FUNCTION_BLOCK FB_SlaveCart
VAR
	
	//Driving force of the car io
	m_driveForce AT %I* :Vec2i;
	
	//stabilizing foot sensor  (normally-closed contact)
	m_stabilizFootSensorLeft AT%I* :BOOL;
	m_stabilizFootSensorRight AT%I* :BOOL;
	m_drivingLeverSensorAuto AT%I* :BOOL;
	m_drivingLeverSensorManual AT%I* :BOOL;
	
	//Trocar IO check
	m_trocarIO AT %I* : ARRAY [1..4] OF UDINT;
	m_trocarCheck : ARRAY [1..4] OF FB_trocarDetect;
	m_trocarFlag : ARRAY [1..4] OF BOOL;
	m_trocarOnFlag : INT:=0;
	
	//output screw break IO 
	m_screwBreak AT %Q* : BOOL;
	m_screwBreakSR : SR;
	
	//car overhang rotation signal is in the arm
	m_carRotaOverhangIO AT%I* : ARRAY [1..4] OF UDINT;
	m_rotaButtonDetect : ARRAY [1..4] OF FB_rotaButtonDetect;
	m_rotaOverhangOnFlag : UDINT :=0;
	
	//cart joint
	m_cartJoints: ARRAY [1..g_cartJntNum] OF FB_CartJoint;
	
	// cart status
	m_cartStatus  : ST_CartStatus;
	
	//cart joint 5 enable detect
	m_standColumnEnableDetect : FB_cartJntEnableDetect;
	m_standColumnDisenableDetect : FB_cartJntDisenableDetect;

	// arm joint data
	m_curMotorPos :Vec8d;
	m_curLinkPos :Vec8d;
	m_curLinkSingle :Vec8d;
	m_curJntPos :Vec8d;
	m_curDHJntPos :Vec6d;
	m_curGripAngle :LREAL;
	m_curJntVel :Vec8d;
	m_curDHJntVel :Vec6d;
	m_curJntTrq :Vec8d;
	m_rawJntCurrent :Vec8d;
	m_filtJntCurrent :Vec8d;
	m_cmdJntTrq :Vec8d;
	m_cmdJntCurrent : Vec8d;
	m_cmdJntPos :Vec8d;
	m_cmdJntVel :Vec8d;

	//SDO Writer
	m_CommunicationCycleInitMZSub1:ARRAY [1..3] OF FB_EcCoESdoWrite;
	m_CommunicationCycleInitMZSub2:ARRAY [1..3] OF FB_EcCoESdoWrite;
	m_CommunicationCycleSub1:INT:=1;
	m_CommunicationCycleSub2:INT:=-3;
	
	//update ui information
	m_joystickSignal:Vec8d;
	m_cartDataFromUI : ST_CartUIData;
	m_ctrlEnable : ST_uiControl;
	m_surgicalStatusF : F_TRIG;
	
	//stand column adjust of setup joint 3
	m_columnJntVel : LREAL;
	m_columnAdjustEnable : BOOL;
	m_limitBufferForCtrl : LREAL := 0.01;
	m_midJntPos : LREAL := 0.1;
	enableTon : ARRAY [1..4] OF FB_TON;
	
	// collision detection
	m_collisionDetection : FB_CartCollisionDetect;
	m_collisionFlag :BOOL:=false;
END_VAR

PROPERTY cartDockingState : UINT
GET
END_GET
SET
m_cartDataFromUI.m_cartDockingState := cartDockingState;
END_SET
END_PROPERTY

PROPERTY cartDrapingState : UINT
GET
END_GET
SET
m_cartDataFromUI.m_cartDrapingState := cartDrapingState;
END_SET
END_PROPERTY

METHOD checkIO : BOOL
VAR_INPUT
END_VAR
VAR
	i:INT;
END_VAR
//check overhang rotation button
m_rotaOverhangOnFlag := MAX( m_rotaButtonDetect[1].run(m_carRotaOverhangIO[1]), m_rotaButtonDetect[2].run(m_carRotaOverhangIO[2]),m_rotaButtonDetect[3].run(m_carRotaOverhangIO[3]),m_rotaButtonDetect[4].run(m_carRotaOverhangIO[4]));

FOR i := 1 TO g_sArmNum BY 1 DO
	//trocar in place monitor
	m_trocarFlag[i] := m_trocarCheck[i].run(m_trocarIO[i] );
END_FOR

m_trocarOnFlag := BOOL_TO_INT(m_trocarFlag[1]) + BOOL_TO_INT(m_trocarFlag[2]) + BOOL_TO_INT(m_trocarFlag[3]) + BOOL_TO_INT(m_trocarFlag[4]);

//setup robot joint 3 adjust and drive column movement
m_columnAdjustEnable :=columnAdjustEnable(o_columnJntVel => m_columnJntVel  );
END_METHOD

PROPERTY cmdJntPos : REFERENCE TO Vec8d
GET
cmdJntPos REF= m_cmdJntPos;
END_GET
END_PROPERTY

PROPERTY cmdJntVel : REFERENCE TO Vec8d
GET
cmdJntVel REF= m_cmdJntVel;
END_GET
END_PROPERTY

METHOD columnAdjustEnable : BOOL
VAR_INPUT
END_VAR

VAR_OUTPUT
	o_columnJntVel : LREAL;
END_VAR

VAR_STAT
	curJntPos : vec4d;
	curJntVel : vec4d;
	columnJntVel : vec4d;
	adjustStartFlag : vec4b;
	m_columnAdjustEnable : vec4b;
END_VAR
VAR
	i : INT;
	armId : INT;
	limitDis : vec4d;
	m_adjustFlag : vec4b;
END_VAR

FOR i := 1 TO g_sArmNum DO
	curJntPos[i] := SetupArmControl.m_setupRobot.m_setupArms[i].m_curJntPos[3];
	curJntVel[i] := SetupArmControl.m_setupRobot.m_setupArms[i].m_curJntVel[3];
	m_adjustFlag[i] := SetupArmControl.m_setupRobot.m_setupArms[i].m_manualAdjustOnFlag AND m_trocarOnFlag=0 AND SetupArmControl.m_setupRobot.m_setupArmState[i] = SetupArmState_ManualAdjust 
									AND NOT SafetyCheck.m_SafetyCheck.m_jntErrFlag[i,0,2] AND NOT SafetyCheck.m_SafetyCheck.m_jntErrFlag[i,0,3] AND NOT SafetyCheck.m_SafetyCheck.m_jntErrFlag[i,3,3] AND NOT SafetyCheck.m_SafetyCheck.m_jntErrFlag[i,2,3] ;
	
	IF m_adjustFlag[i] THEN
		limitDis[i] := MIN(GVL_SetupMotorParameters.g_maxJntPos[i,3] - curJntPos[i], curJntPos[i]-GVL_SetupMotorParameters.g_minJntPos[i,3]);
		IF limitDis[i] < m_limitBufferForCtrl THEN
			adjustStartFlag[i] := TRUE; 
			columnJntVel[i] := sign(m_midJntPos - curJntPos[i]) * GVL_CartControlParameters.g_maxJntVel[5];
		
		ELSIF limitDis[i] >= m_limitBufferForCtrl AND NOT m_columnAdjustEnable[i] THEN
			columnJntVel[i] := 0;
			adjustStartFlag[i] := FALSE;
			
		ELSE
			IF curJntVel[i] <> 0 AND adjustStartFlag[i] THEN
				columnJntVel[i] := -LIMIT(-GVL_CartControlParameters.g_maxJntVel[5], curJntVel[i], GVL_CartControlParameters.g_maxJntVel[5]);
			END_IF
		END_IF
		
		armId := i;
		enableTon[i](IN:= adjustStartFlag[i], PT:= T#3S, Q=> m_columnAdjustEnable[i], ET=> );
		EXIT;
	ELSE
		adjustStartFlag[i] := FALSE;
		columnJntVel[i] := 0;
	END_IF
	enableTon[i](IN:= adjustStartFlag[i], PT:= T#3S, Q=> m_columnAdjustEnable[i], ET=> );
END_FOR

//output stand column joint velocity and start adjust single
IF armId > 0 THEN
	o_columnJntVel := columnJntVel[armId];
END_IF
columnAdjustEnable := m_columnAdjustEnable[1] OR m_columnAdjustEnable[2] OR m_columnAdjustEnable[3] OR m_columnAdjustEnable[4];
END_METHOD

PROPERTY ctrlEnable : REFERENCE TO ST_uiControl
GET
ctrlEnable REF= m_ctrlEnable;
END_GET
SET
END_SET
END_PROPERTY

PROPERTY curDHJntPos :REFERENCE TO Vec6d
GET
curDHJntPos ref= m_curDHJntPos;
END_GET
END_PROPERTY

PROPERTY curDHJntVel :REFERENCE TO Vec6d
GET
curDHJntVel REF= m_curDHJntVel;
END_GET
END_PROPERTY

PROPERTY curJntCurrent :REFERENCE TO Vec8d
GET
curJntCurrent ref=m_filtJntCurrent;
END_GET
END_PROPERTY

PROPERTY curJntPos : REFERENCE TO Vec8d
GET
curJntPos ref=m_curJntPos;
END_GET
END_PROPERTY

PROPERTY curJntVel :REFERENCE TO Vec8d
GET
curJntVel ref=m_curJntVel;
END_GET
END_PROPERTY

PROPERTY curLinkPos :REFERENCE TO Vec8d
GET
curLinkPos ref=m_curLinkPos;
END_GET
END_PROPERTY

PROPERTY curMotorPos : REFERENCE TO  Vec8d
GET
curMotorPos ref=m_curMotorPos;
END_GET
END_PROPERTY

METHOD PUBLIC enable : BOOL
VAR_IN_OUT CONSTANT
	i_jntIdx :Vec8i;
END_VAR
VAR
	i :INT ;
END_VAR
FOR i:=1 TO g_cartJntNum DO
	IF 3<=i AND i<5 THEN
		IF 1= i_jntIdx[i] THEN
			m_cartJoints[i].enableMZ();
		ELSE
			m_cartJoints[i].disable();
		END_IF
	ELSIF i = 5 THEN
		IF 1= i_jntIdx[i] THEN
			m_screwBreak := m_standColumnEnableDetect.run(IOValue:= m_cartJoints[i].enableMZ());
			m_standColumnDisenableDetect.run(IOValue:=FALSE );
		ELSE
			m_standColumnEnableDetect.run(IOValue:= FALSE);
			m_screwBreak :=  NOT m_standColumnDisenableDetect.run(IOValue:=m_cartJoints[i].disable());
		END_IF
	ELSE
		IF 1= i_jntIdx[i] THEN
			m_cartJoints[i].enable();
		ELSE
			m_cartJoints[i].disable();
		END_IF
	END_IF
END_FOR
END_METHOD

METHOD init : BOOL
VAR_INPUT
END_VAR
VAR
	i:INT;
END_VAR


// cart joint init
FOR i:= 1 TO g_cartJntNum BY 1 DO
	m_cartJoints[i].init(i, g_cartCtrlCycleTime);
END_FOR


// joint init
FOR i:=1 TO g_cartJntNum DO
	m_cartJoints[i].initJntPos();
END_FOR


// update cart status if joint position is re-init
updateStatus();



//MingZhi drive example Initialize the communication period
FOR i := 1 TO 3 BY 1 DO
	m_CommunicationCycleInitMZSub1[i](sNetID:= GVL_CartJointEncoderCaliData.g_slaveCartNetID,
				nSlaveAddr := GVL_CartJointEncoderCaliData.g_slaveCartJointNetPort[i+2],
				nSubIndex:=1,nIndex:=16#60C2,pSrcBuf:=ADR(m_CommunicationCycleSub1),cbBufLen:=SIZEOF(m_CommunicationCycleSub1),bExecute:=TRUE);
	
	IF NOT m_CommunicationCycleInitMZSub1[i].bBusy THEN
		m_CommunicationCycleInitMZSub1[i](bExecute:=FALSE);
	END_IF
					
	m_CommunicationCycleInitMZSub2[i](sNetID:= GVL_CartJointEncoderCaliData.g_slaveCartNetID,
					nSlaveAddr := GVL_CartJointEncoderCaliData.g_slaveCartJointNetPort[i+2],
					nSubIndex:=2,nIndex:=16#60C2,pSrcBuf:=ADR(m_CommunicationCycleSub2),cbBufLen:=SIZEOF(m_CommunicationCycleSub2),bExecute:=TRUE);
	
	IF NOT m_CommunicationCycleInitMZSub2[i].bBusy THEN
		m_CommunicationCycleInitMZSub2[i](bExecute:=FALSE);
	END_IF
END_FOR
END_METHOD

METHOD  joystickSignalAnalysis : Vec8d 
VAR_INPUT
	i_joystickDataFromUI:ARRAY [0..21] OF USINT;
END_VAR

VAR_STAT
	i:INT;
	m_handData:ARRAY [0..21] OF USINT;
	m_outHandData : Vec8d;
END_VAR

IF i_joystickDataFromUI[0] = 16#FF THEN
	m_handData := i_joystickDataFromUI;
	m_outHandData[1] :=m_handData[7]*256 + m_handData[8]; // car  joint5 pillar
	m_outHandData[2] :=m_handData[3]*256 + m_handData[4]; //car joint7 beamStretch
	m_outHandData[3] :=m_handData[1]*256 + m_handData[2]; // car joint6  beamRot
	m_outHandData[4] :=m_handData[5]*256 + m_handData[6]; // joint8 overhang 
	m_outHandData[5] :=m_handData[9]*256 + m_handData[10];
	m_outHandData[6] :=m_handData[11]*256 + m_handData[12];
	m_outHandData[7] :=m_handData[13]*256 + m_handData[14];
	m_outHandData[8] :=m_handData[15]*256 + m_handData[16];
END_IF
joystickSignalAnalysis:=m_outHandData;
END_METHOD

METHOD ProcessingUIData : BOOL
VAR_IN_OUT CONSTANT
	//UI information, import from UI controller
	i_UIData :ST_CartUIData;
END_VAR
VAR
	i : INT;
END_VAR
m_joystickSignal := joystickSignalAnalysis(i_UIData.m_joystickDataFromUI);

m_ctrlEnable:=i_UIData.m_ctrlEnableFromUI;

m_cartDataFromUI.m_standColumnHightLimit := i_UIData.m_standColumnHightLimit;

m_cartDataFromUI.m_cartSpecificPosDraping := GVL_CartControlParameters.g_surgicalDrapingPos;

FOR i := 1 TO g_sArmNum BY 1 DO
	IF i_UIData.m_surgicalSite > 0 AND i_UIData.m_surgicalLocation > 0 THEN
		m_cartDataFromUI.m_cartSpecificPosDocking[i + 4] := GVL_CartControlParameters.g_surgicalOrientPos[i_UIData.m_surgicalSite, i_UIData.m_surgicalLocation,i];
	END_IF
END_FOR

m_surgicalStatusF(CLK:= GVL_interactUI.g_surgicalStatus , Q=> );
IF m_surgicalStatusF.Q THEN
	cartDrapingState := 0;
END_IF

IF NOT (m_cartDataFromUI.m_surgicalSite = i_UIData.m_surgicalSite) OR NOT (m_cartDataFromUI.m_surgicalLocation = i_UIData.m_surgicalLocation) THEN
	cartDockingState := 0;
END_IF

m_cartDataFromUI.m_surgicalSite := i_UIData.m_surgicalSite;
m_cartDataFromUI.m_surgicalLocation := i_UIData.m_surgicalLocation;
END_METHOD

PROPERTY status : ST_CartStatus
GET
status := m_cartStatus;
END_GET
END_PROPERTY

METHOD PUBLIC updateCmds : BOOL
VAR_IN_OUT CONSTANT
	i_cartCtrlCmd : ST_SlaveArmCtrlCmds;
END_VAR
VAR
	i:INT;
END_VAR
m_cmdJntTrq:=i_cartCtrlCmd.m_cmdJntTrq;
m_cmdJntPos :=i_cartCtrlCmd.m_cmdJntPos;
m_cmdJntVel :=i_cartCtrlCmd.m_cmdJntVel;


// enable/disable joints
enable(i_cartCtrlCmd.m_jntEnableFlag);

// position/Velocity control
FOR i:=1 TO g_sJntNum DO 
	IF i_cartCtrlCmd.m_jntOPMode[i]=DriverOPMode_Pos THEN
		m_cmdJntTrq[i]:=0;
		m_cmdJntVel[i]:=0;
		m_cartJoints[i].updateCmd(DriverOPMode_Pos,m_cmdJntPos[i],m_cmdJntTrq[i],m_cmdJntVel[i]);
	ELSIF i_cartCtrlCmd.m_jntOPMode[i]=DriverOPMode_Vel THEN
		m_cmdJntTrq[i]:=0;
		m_cmdJntPos[i]:=0;
		m_cartJoints[i].updateCmd(DriverOPMode_Pos,m_cmdJntPos[i],m_cmdJntTrq[i],m_cmdJntVel[i]);
	ELSIF i_cartCtrlCmd.m_jntOPMode[i]=DriverOPMode_MZPos  THEN
		m_cmdJntTrq[i]:=0;
		m_cmdJntVel[i]:=0;
		//Input torque mode because the operating mode word for the contour position mode of the MingZhi driver is 1
		m_cartJoints[i].updateCmd(DriverOPMode_Trq,m_cmdJntPos[i],m_cmdJntTrq[i],m_cmdJntVel[i]);
	ELSIF i_cartCtrlCmd.m_jntOPMode[i]=DriverOPMode_cspMZ  THEN
		 m_cartJoints[i].updateCmd(DriverOPMode_cspMZ,m_cmdJntPos[i],m_cmdJntTrq[i],m_cmdJntVel[i]);
	ELSIF DriverOPMode_csvMZ = i_cartCtrlCmd.m_jntOPMode[i] THEN
		m_cartJoints[i].updateCmd(DriverOPMode_csvMZ,m_cmdJntPos[i],m_cmdJntTrq[i],m_cmdJntVel[i]);
	END_IF
END_FOR

// collision check
m_collisionFlag := m_collisionDetection.run(m_rawJntCurrent, m_cmdJntPos, m_curJntVel);
END_METHOD

METHOD PUBLIC updateStatus : BOOL
VAR_INPUT
END_VAR
VAR
	i:INT;
END_VAR
// update joint data
FOR i:=1 TO g_sJntNum DO
	m_cartJoints[i].updateStatus();
END_FOR

//IO output   Horizontal laser IO output   Cross laser IO output
checkIO();


// get joint data
FOR i:=1 TO g_cartJntNum DO
	m_curMotorPos[i]:=m_cartJoints[i].motorPos;
	m_curLinkPos[i]:=m_cartJoints[i].linkPos;
	m_curLinkSingle[i]:=m_cartJoints[i].linkSingle;
	m_curJntPos[i]:=m_cartJoints[i].jntPos;
	m_curJntVel[i]:=m_cartJoints[i].jntVel;
	m_curJntTrq[i]:=m_cartJoints[i].jntTrq;
	m_rawJntCurrent[i]:=m_cartJoints[i].rawCurrent;
	m_filtJntCurrent[i]:=m_cartJoints[i].filtCurrent;
	m_cmdJntCurrent[i]:=m_cartJoints[i].cmdCurrent;
END_FOR
END_METHOD

END_FUNCTION_BLOCK

(* stored: Version 1.1.0.1, ProductVersion 3.1.4024.12
   POU FB_SlaveCart: Id {05baaa0e-c853-48bc-a37c-d593cfa5bf2b}, SpecialFunc None
   Folder property: Id {37b9f91a-fbe1-4cae-807d-574d49e247d7}
   Property cartDockingState: Id {86905c60-a5d0-40a0-947e-e9a92fd9b4c8}
   Get Get: Id {3efac307-74e7-471b-94d7-c9501d69aa9a}
   Set Set: Id {bf6dd221-7fd9-4ea6-9329-7f9485725c41}
   Property cartDrapingState: Id {392660e0-52e3-4ef4-92d3-ba7eba8dd842}
   Get Get: Id {53a9b4f0-7c5c-465f-b7e2-ee69519178b0}
   Set Set: Id {daf76773-35cc-41c7-b97d-fe69cd27cb90}
   Method checkIO: Id {52184f86-1fa7-432c-a16c-6b035dc3943c}
   Property cmdJntPos: Id {488d680a-8342-457b-a395-401f6b755b10}
   Get Get: Id {68835cd8-1473-432f-b232-4a0619dd88bf}
   Property cmdJntVel: Id {7d24481c-3787-4c6e-8b42-03fddb05fef4}
   Get Get: Id {05aa5687-796c-4a75-92d5-951df467cfd7}
   Method columnAdjustEnable: Id {4b81e009-8b8f-44ae-b179-17501f5dd10b}
   Property ctrlEnable: Id {a3baaf86-b572-478d-828a-8abd1832149b}
   Get Get: Id {088e36f0-64b1-4fec-9db7-8ed59d586fe5}
   Set Set: Id {3a6445f6-98f8-4080-a3fd-ced7b89e6f2e}
   Property curDHJntPos: Id {ba1ee581-e55e-41ad-87dc-7b501fc90eb2}
   Get Get: Id {3d3679c2-ef2a-4f6d-a4df-07b6a1b00143}
   Property curDHJntVel: Id {51c1a699-c808-4814-84f2-b43538048e3e}
   Get Get: Id {d647fd51-76de-4dd3-b960-cf5d1f37cc4f}
   Property curJntCurrent: Id {c06954b9-7d46-4bb1-b769-226d7700f290}
   Get Get: Id {803fed64-c7fc-4f5a-a733-13664a3be1b6}
   Property curJntPos: Id {099d6b43-b820-44e6-bf10-79fd50adb0cd}
   Get Get: Id {e95536de-e76f-49e9-afca-f73fdd1cbab0}
   Property curJntVel: Id {4d944a37-47d9-4fd3-a0c1-6a8e3ecf8054}
   Get Get: Id {fe80b852-647f-4f4f-8f1d-7e8c0086b108}
   Property curLinkPos: Id {dd6e8dac-cec3-48df-b41e-0a55e5f7b25c}
   Get Get: Id {68094696-79da-4c76-8f41-c8adfd451a61}
   Property curMotorPos: Id {4d7df53d-6ac0-4195-b87b-e20244051d14}
   Get Get: Id {61be3c14-3c98-4743-b66a-f89744318c7b}
   Method enable: Id {b1f8fb89-f8ac-43fc-a9cf-b5c213a4b36e}
   Method init: Id {a9830b95-e937-4a29-b70e-785e20452d37}
   Method joystickSignalAnalysis: Id {15b803f9-93d6-4377-9b18-7562f2015d41}
   Method ProcessingUIData: Id {217a26c8-8c06-4704-8681-3cd189d05dd8}
   Property status: Id {cd2a750f-147a-42a5-85cd-a7d5a815c963}
   Get Get: Id {c1788322-40e1-4e3e-a26b-a8239c1e1e6d}
   Method updateCmds: Id {a083537e-6f52-4b88-8b83-3c9a5d0db87a}
   Method updateStatus: Id {7dc0698e-0910-43df-8937-4fb176791915} *)
